FUNCTION_BLOCK FB_ModifyAutomaticControlSettings
VAR_INPUT
	stParamOpenLoopControllSettings 	: REFERENCE TO ST_OpenLoopControlSettings;
	stParamClosedLoopControllSettings 	: REFERENCE TO ST_ClosedLoopControlSettings;
	stModify 							: ST_ModifyAutomaticControlSettings;
END_VAR
VAR_OUTPUT
END_VAR
VAR
END_VAR

IF stModify.bSetNewMaxFlowCapacity THEN
	stParamOpenLoopControllSettings.fMaxFlowCapacity := stModify.fNewMaxFlowCapacity;
	stModify.bSetNewMaxFlowCapacity := FALSE;
END_IF

IF stModify.bSetNewProportionalGain THEN
	stParamClosedLoopControllSettings.fProportionalGain := stModify.fNewProportionalGain;
	stModify.bSetNewProportionalGain := FALSE;
END_IF

IF stModify.bSetNewIntegralGain THEN
	stParamClosedLoopControllSettings.fIntegralGain := stModify.fNewIntegralGain;
	stModify.bSetNewIntegralGain := FALSE;
END_IF

IF stModify.bSetNewMaxPositionError THEN
	stParamClosedLoopControllSettings.fMaxPositionError:= stModify.fNewMaxPositionError;
	stModify.bSetNewMaxPositionError := FALSE;
END_IF

END_FUNCTION_BLOCK

(* stored: Version 1.1.0.1, ProductVersion 3.1.4024.11
   POU FB_ModifyAutomaticControlSettings: Id {b10fa07f-8b07-44ec-993b-317e37a0c116}, SpecialFunc None *)
